# EPICS substitutions: elioApp/Db/EL4038.substitutions
file EL4038.template { pattern
{ CHAN	}
{ 1	}
{ 2	}
{ 3	}
{ 4	}
{ 5	}
{ 6	}
{ 7	}
{ 8	}
}
